FUNCTION Convert_BOOL_TO_STRING : BOOL
VAR_INPUT
	in : BOOL;
	out : REFERENCE TO STRING;
END_VAR

out := BOOL_TO_STRING(in);
Convert_BOOL_TO_STRING := TRUE;

END_FUNCTION

(* stored: Version 1.1.0.1, ProductVersion 3.1.4024.12
   POU Convert_BOOL_TO_STRING: Id {3e44b2f9-f372-4a1d-97e6-e162a3bec77b}, SpecialFunc None *)
